ABB RAPID module: TargetPoint_Robot.modx

MODULE Tesi_Lorenzo

    LOCAL PERS tooldata gripper:=[TRUE,[[0,0,117.85],[0.966,0,0,0.259]],[0.59,[0.15,0.01,57.98],[1,0,0,0],0,0,0]];

    LOCAL CONST robtarget HomePose:=[[-417.51,304.76,527.54],[0.04416,-0.99506,0.05359,0.07092],[1,-1,-1,0],[9000000000,9000000000,9000000000,9000000000,9000000000,9000000000]];

    LOCAL CONST robtarget GP_S1:=[[-587.53,81.71,80.00],[0.00266,-0.71165,-0.70252,0.00450],[1,-1,-1,0],[9000000000,9000000000,9000000000,9000000000,9000000000,9000000000]];
    LOCAL CONST robtarget GP_S2:=[[-495.42,82.83,79.70],[0.00270,-0.71180,-0.70234,0.00463],[1,-1,-1,0],[9000000000,9000000000,9000000000,9000000000,9000000000,9000000000]];
    LOCAL CONST robtarget GP_S3:=[[-409.29,79.69,79.70],[0.00287,-0.71167,-0.70249,0.00485],[1,-1,-1,0],[9000000000,9000000000,9000000000,9000000000,9000000000,9000000000]];
    LOCAL CONST robtarget CTR_SCREW_S:=[[-331.81,67.31,109.41],[0.01684,-0.99967,0.01901,0.00405],[1,-1,-1,0],[9000000000,9000000000,9000000000,9000000000,9000000000,9000000000]];
    LOCAL CONST robtarget CTR_S1:=[[-376.88,145.90,108.27],[0.00337,-0.71197,-0.70219,0.00486],[1,-1,-1,0],[9000000000,9000000000,9000000000,9000000000,9000000000,9000000000]];

    LOCAL CONST robtarget GP_R1:=[[-518.29,290.98,80.71],[0.00241,-0.71171,-0.70245,0.00453],[1,-1,-1,0],[9000000000,9000000000,9000000000,9000000000,9000000000,9000000000]];
    LOCAL CONST robtarget GP_R2:=[[-517.64,389.63,80.91],[0.00241,-0.71171,-0.70245,0.00453],[1,-1,-1,0],[9000000000,9000000000,9000000000,9000000000,9000000000,9000000000]];
    LOCAL CONST robtarget GP_SCREWDRIVER:=[[-610.34,380.34,81.06],[0.00188,-0.71177,-0.70240,0.00441],[1,-1,-1,0],[9000000000,9000000000,9000000000,9000000000,9000000000,9000000000]];
    LOCAL CONST robtarget GP_R3:=[[-518.10,490.01,81.19],[0.00241,-0.71171,-0.70245,0.00456],[1,-1,-1,0],[9000000000,9000000000,9000000000,9000000000,9000000000,9000000000]];
    LOCAL CONST robtarget GP_R4:=[[-429.89,340.60,80.02],[0.00241,-0.71203,-0.70213,0.00456],[1,-1,-1,0],[9000000000,9000000000,9000000000,9000000000,9000000000,9000000000]];
    LOCAL CONST robtarget GP_R5:=[[-429.33,440.59,79.86],[0.00241,-0.71196,-0.70220,0.00456],[1,-1,-1,0],[9000000000,9000000000,9000000000,9000000000,9000000000,9000000000]];
    LOCAL CONST robtarget CTR_SCREW_R:=[[-376.19,301.83,108.40],[0.00297,-0.71167,-0.70245,0.00456],[1,-1,-1,0],[9000000000,9000000000,9000000000,9000000000,9000000000,9000000000]];
    LOCAL CONST robtarget CTR_R1:=[[-375.88,456.32,113.78],[0.00249,-0.71171,-0.70245,0.00456],[1,-1,-1,0],[9000000000,9000000000,9000000000,9000000000,9000000000,9000000000]];


ENDMODULE
